PROGRAM robotCall
VAR

	robotCommsInstance: FB_RobotComms;
END_VAR

VAR PERSISTENT
	
END_VAR

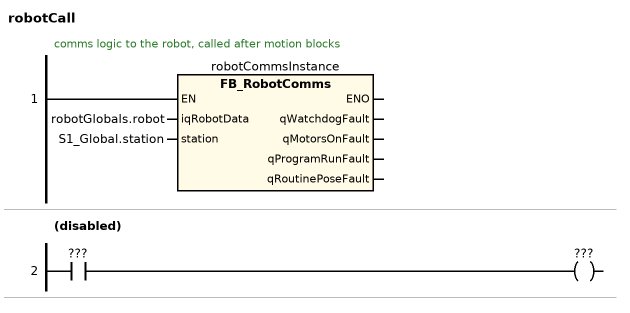
// NETWORK 1
// comms logic to the robot, called after motion blocks
robotCommsInstance(iqRobotData := robotGlobals.robot, station := S1_Global.station); // FB_RobotComms

// NETWORK 2 (disabled)
// ??? := ???;

END_PROGRAM

(* stored: Version 1.1.0.1, ProductVersion 3.1.4024.11
   POU robotCall: Id {db02258e-4bcf-4f9a-ac9f-2be537a76e6c}, SpecialFunc None *)
